FUNCTION_BLOCK CruiseManager (* Manages the state of the cruise control *)
  (* Standard: 61499-2 *)
  (* Version 0.2, 2003-12-04, JHC, Rockwell Automation, Renamed for better indexing. *)
  (* Version 0.1, 2002-11-05, JHC, Rockwell Automation, Corrected missing ST element in Algorithm REQ. *)
  (* Version 0.0, 2000-05-30, JHC, Rockwell Automation *)
  (* Compiler header: package fb.rt.benchmarks.cruisecontrol; *)
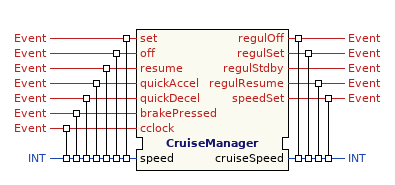
  EVENT_INPUT
    set WITH speed;
    off WITH speed;
    resume WITH speed;
    quickAccel WITH speed; (* increase desired speed by 5km/h *)
    quickDecel WITH speed;
    brakePressed WITH speed;
    cclock WITH speed; (* 10ms tick *)
  END_EVENT
  EVENT_OUTPUT
    regulOff WITH cruiseSpeed;
    regulSet WITH cruiseSpeed;
    regulStdby;
    regulResume WITH cruiseSpeed;
    speedSet WITH cruiseSpeed;
  END_EVENT
  VAR_INPUT
    speed : INT := 0;
  END_VAR
  VAR_OUTPUT
    cruiseSpeed : INT := 0;
  END_VAR
  VAR
    desiredSpeed : int := 0;
  END_VAR
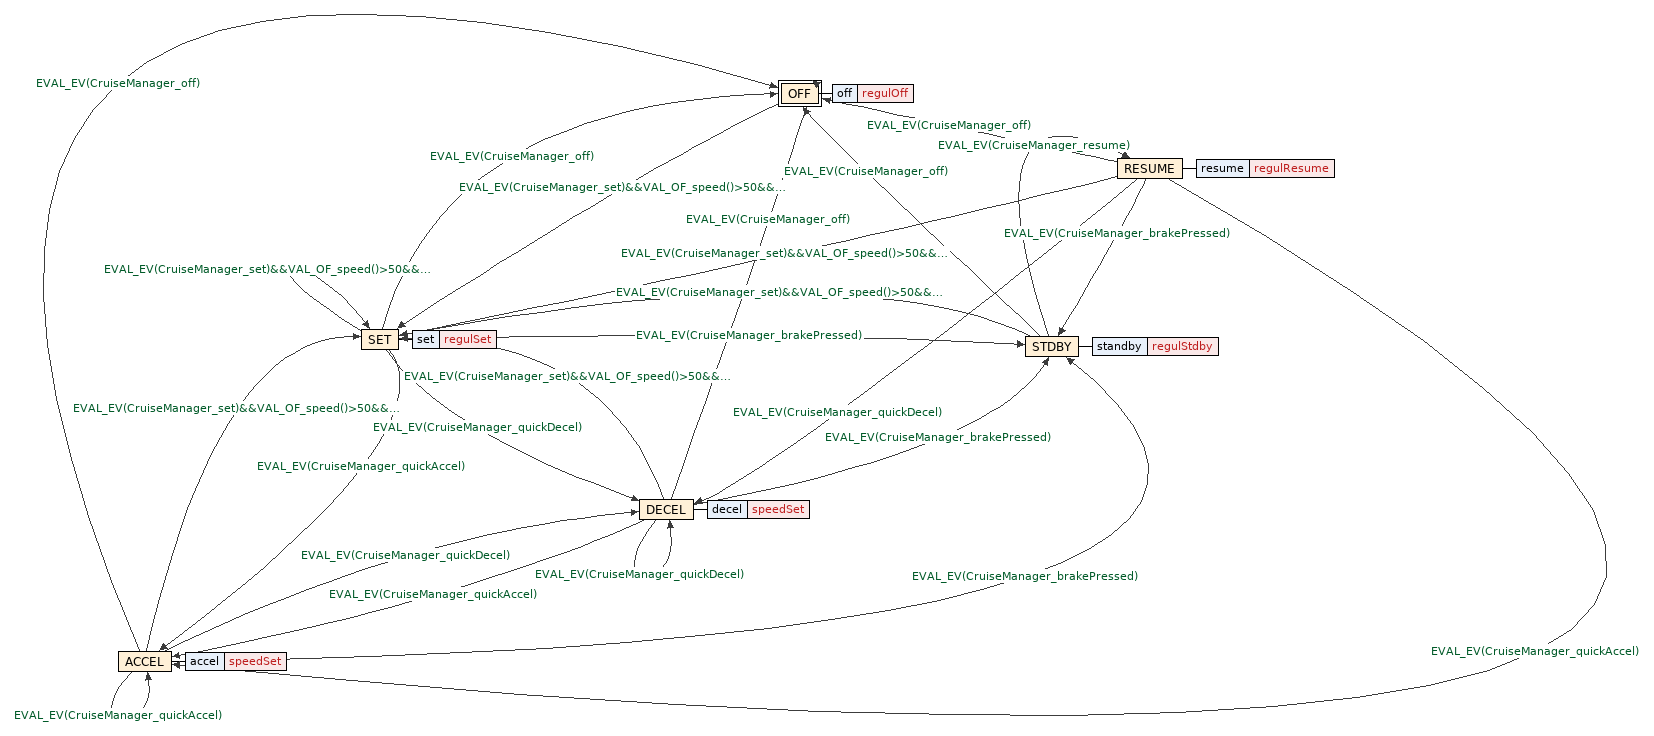
  EC_STATES
    OFF : off -> regulOff; (* Initial State *)
    SET : set -> regulSet;
    STDBY : standby -> regulStdby;
    RESUME : resume -> regulResume;
    ACCEL : accel -> speedSet;
    DECEL : decel -> speedSet;
  END_STATES
  EC_TRANSITIONS
    OFF TO SET := EVAL_EV(CruiseManager_set)&&VAL_OF_speed()>50&&VAL_OF_speed()<170;
    SET TO OFF := EVAL_EV(CruiseManager_off);
    SET TO SET := EVAL_EV(CruiseManager_set)&&VAL_OF_speed()>50&&VAL_OF_speed()<170;
    SET TO STDBY := EVAL_EV(CruiseManager_brakePressed);
    SET TO ACCEL := EVAL_EV(CruiseManager_quickAccel);
    SET TO DECEL := EVAL_EV(CruiseManager_quickDecel);
    STDBY TO OFF := EVAL_EV(CruiseManager_off);
    STDBY TO SET := EVAL_EV(CruiseManager_set)&&VAL_OF_speed()>50&&VAL_OF_speed()<170;
    STDBY TO RESUME := EVAL_EV(CruiseManager_resume);
    RESUME TO OFF := EVAL_EV(CruiseManager_off);
    RESUME TO SET := EVAL_EV(CruiseManager_set)&&VAL_OF_speed()>50&&VAL_OF_speed()<170;
    RESUME TO STDBY := EVAL_EV(CruiseManager_brakePressed);
    RESUME TO ACCEL := EVAL_EV(CruiseManager_quickAccel);
    RESUME TO DECEL := EVAL_EV(CruiseManager_quickDecel);
    ACCEL TO OFF := EVAL_EV(CruiseManager_off);
    ACCEL TO SET := EVAL_EV(CruiseManager_set)&&VAL_OF_speed()>50&&VAL_OF_speed()<170;
    ACCEL TO STDBY := EVAL_EV(CruiseManager_brakePressed);
    ACCEL TO ACCEL := EVAL_EV(CruiseManager_quickAccel);
    ACCEL TO DECEL := EVAL_EV(CruiseManager_quickDecel);
    DECEL TO OFF := EVAL_EV(CruiseManager_off);
    DECEL TO SET := EVAL_EV(CruiseManager_set)&&VAL_OF_speed()>50&&VAL_OF_speed()<170;
    DECEL TO STDBY := EVAL_EV(CruiseManager_brakePressed);
    DECEL TO ACCEL := EVAL_EV(CruiseManager_quickAccel);
    DECEL TO DECEL := EVAL_EV(CruiseManager_quickDecel);
  END_TRANSITIONS
  ALGORITHM off IN ST:
desiredSpeed= 0;
VAL_OF_cruiseSpeed()= 0;
  END_ALGORITHM
  ALGORITHM set IN ST:
desiredSpeed= VAL_OF_speed();
VAL_OF_cruiseSpeed()= desiredSpeed;
  END_ALGORITHM
  ALGORITHM resume IN ST:
VAL_OF_cruiseSpeed()= desiredSpeed;
  END_ALGORITHM
  ALGORITHM standby IN ST:
VAL_OF_cruiseSpeed()= 0;
  END_ALGORITHM
  ALGORITHM accel IN ST:
if( desiredSpeed < 165) {
    desiredSpeed= desiredSpeed + 5;
    VAL_OF_cruiseSpeed()= desiredSpeed;
};
  END_ALGORITHM
  ALGORITHM decel IN ST:
if (desiredSpeed >= 5) {
    desiredSpeed= desiredSpeed - 5;
    VAL_OF_cruiseSpeed()= desiredSpeed;
}else{ desiredSpeed= 0;
 };
  END_ALGORITHM
END_FUNCTION_BLOCK
